PROGRAM PrgMqttCom
VAR
	fbMqttClient : FB_IotMqttClient;
	bSetParameter : BOOL := TRUE;
	bConnect : BOOL := TRUE;
	
	(* published message *)
	sTopicPub : STRING(255) := 'MyTopic';
	sPayloadPub : STRING(255);
	i: UDINT;
	fbTimer : TON := (PT:=T#1S);
	
	(* received message *)
	bSubscribed : BOOL;
	sTopicSub : STRING(255) := 'MyTopic';
	{attribute 'TcEncoding':='UTF-8'}
	sTopicRcv : STRING(255);
	{attribute 'TcEncoding':='UTF-8'}
	sPayloadRcv : STRING(255);
	fbMessageQueue : FB_IotMqttMessageQueue;
	fbMessage : FB_IotMqttMessage;
	
	hrErrorOccurred : HRESULT; // contains the latest occurred error
END_VAR

IF bSetParameter THEN
	bSetParameter := FALSE;
	fbMqttClient.sHostName:= 'localhost';
	fbMqttClient.nHostPort:= 1883;
//	fbMqttClient.sClientId:= 'MyTcMqttClient'; 
	fbMqttClient.sTopicPrefix:= ''; 
//	fbMqttClient.nKeepAlive:= 60; 
//	fbMqttClient.sUserName:= ;
//	fbMqttClient.sUserPassword:= ; 
//	fbMqttClient.stWill:= ; 
//	fbMqttClient.stTLS:= ;
	fbMqttClient.ipMessageQueue := fbMessageQueue;
END_IF

fbMqttClient.Execute(bConnect);
IF fbMqttClient.bError THEN
	// add your error logging here
	hrErrorOccurred := fbMqttClient.hrErrorCode;
END_IF

IF fbMessageQueue.nQueuedMessages > 0 THEN
	IF fbMessageQueue.Dequeue(fbMessage:=fbMessage) THEN
		fbMessage.GetTopic(pTopic:=ADR(sTopicRcv), nTopicSize:=SIZEOF(sTopicRcv) );
		fbMessage.GetPayload(pPayload:=ADR(sPayloadRcv), nPayloadSize:=SIZEOF(sPayloadRcv), bSetNullTermination:=FALSE);
	END_IF
END_IF

IF fbMqttClient.bConnected THEN
	IF NOT bSubscribed THEN
		bSubscribed := fbMqttClient.Subscribe(sTopic:=sTopicSub, eQoS:=TcIotMqttQos.AtMostOnceDelivery);
		IF fbMqttClient.bError THEN
			// add your error logging here
			hrErrorOccurred := fbMqttClient.hrErrorCode;
		END_IF
	END_IF
	fbTimer(IN:=TRUE);
	IF fbTimer.Q THEN // publish new payload every second
		fbTimer(IN:=FALSE);
		i := i + 1;
		sPayloadPub := CONCAT('MyMessage', TO_STRING(i));
		fbMqttClient.Publish(	sTopic:= sTopicPub, 
								pPayload:= ADR(sPayloadPub), nPayloadSize:= LEN2(ADR(sPayloadPub))+1, 
								eQoS:= TcIotMqttQos.AtMostOnceDelivery, bRetain:= FALSE, bQueue:= FALSE );
		IF fbMqttClient.bError THEN
			// add your error logging here
			hrErrorOccurred := fbMqttClient.hrErrorCode;
		END_IF
	END_IF
END_IF

END_PROGRAM

(* stored: Version 1.1.0.1
   POU PrgMqttCom: Id {c70f107a-6ca5-4bfb-b775-e2929cbf9dae}, SpecialFunc None *)
